(* Schneider Machine Expert - Basic project punya faris yang diomelin Ichsan Pan8, file version 1.7.0.0 *)
(* ProjectInformations: Name=New project *)

HARDWARE
  Cpu 0: TM221M16R/G
  EthernetConfiguration: NetworkName=M221, IpAllocationMode=FixedAddress, IpAddress=0.0.0.0, SubnetMask=0.0.0.0
  SerialLineConfiguration: Baud=Baud19200, Parity=ParityEven, DataBits=DataBits8, StopBits=StopBits1, PhysicalMedium=PhysicalMediumRs485, TransmissionMode=TransmissionModeModbusRtu, SlaveId=1, Addressing=SlaveAddressing
  MastTask: UsePeriodScanMode=false, PeriodScan=100
  FastTask: Period=255
  CpuBehavior: StartingMode=StartAsPreviousState, AutoSaveRamOnEeprom=true, WatchdogPeriod=250

SYMBOLS  (address, symbol, comment, settings)
  %M0         "manual"
  %M7         "auto"
  %I0.0       "Selektor"
  %I0.1       "SWITCH MANUAL"
  %I0.2       "Switch1"
  %I0.3       "Switch2"
  %I0.4       "Swutch3"
  %Q0.1       "Lampu1"
  %Q0.2       "Lampu2"

POU New POU
  (* SectionNumber=1 *)

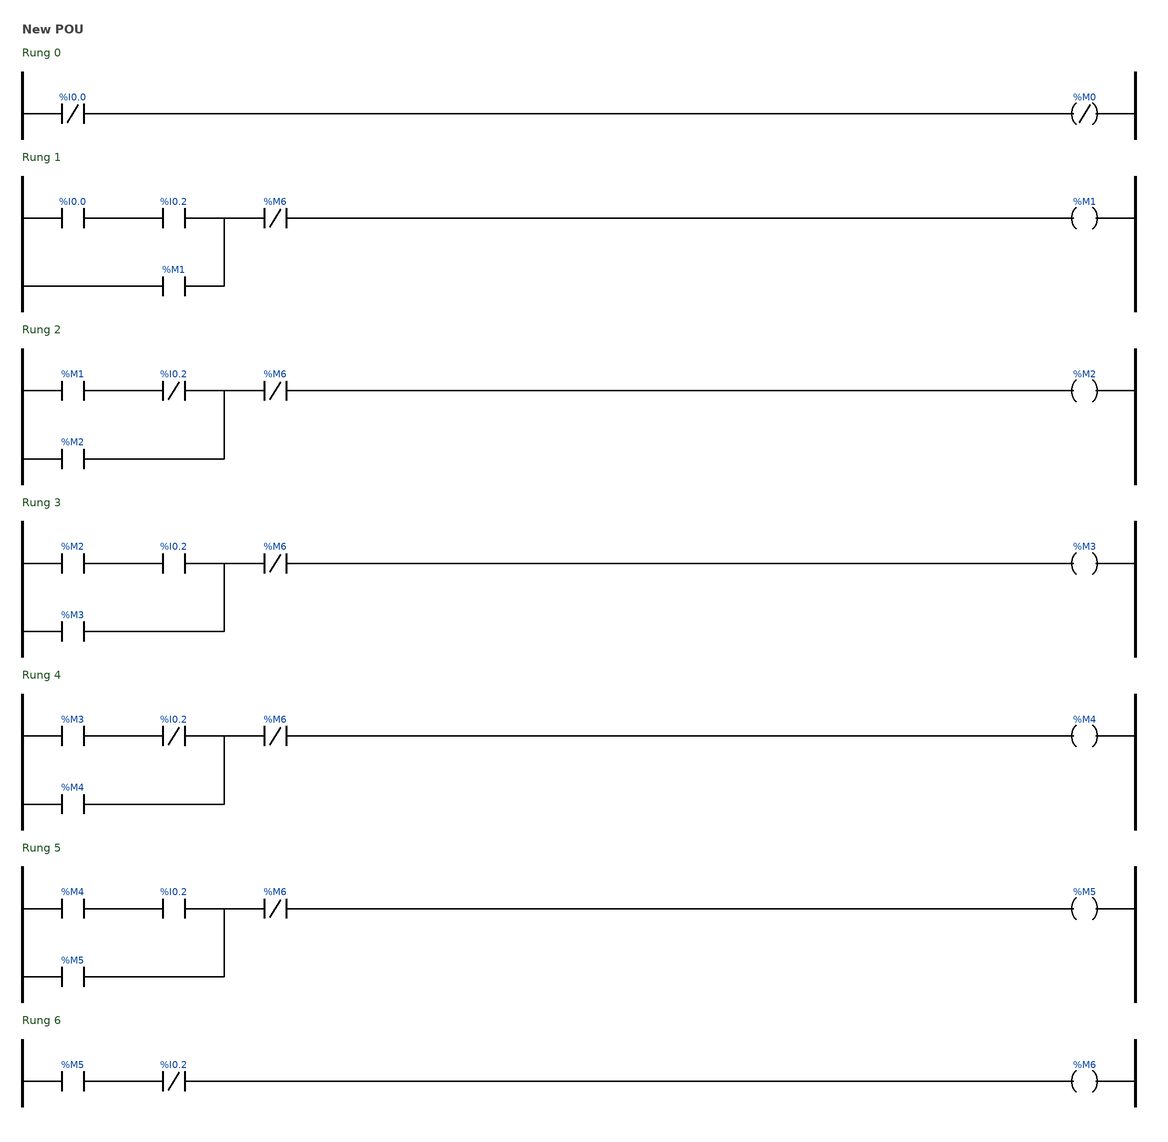

// Rung 0
  LDN %I0.0
  STN %M0
  // as ST:
  //   %M0 := NOT (NOT %I0.0);

// Rung 1
  LD %I0.0
  AND %I0.2
  OR %M1
  ANDN %M6
  ST %M1
  // as ST:
  //   %M1 := (%I0.0 AND %I0.2 OR %M1) AND NOT %M6;

// Rung 2
  LD %M1
  ANDN %I0.2
  OR %M2
  ANDN %M6
  ST %M2
  // as ST:
  //   %M2 := (%M1 AND NOT %I0.2 OR %M2) AND NOT %M6;

// Rung 3
  LD %M2
  AND %I0.2
  OR %M3
  ANDN %M6
  ST %M3
  // as ST:
  //   %M3 := (%M2 AND %I0.2 OR %M3) AND NOT %M6;

// Rung 4
  LD %M3
  ANDN %I0.2
  OR %M4
  ANDN %M6
  ST %M4
  // as ST:
  //   %M4 := (%M3 AND NOT %I0.2 OR %M4) AND NOT %M6;

// Rung 5
  LD %M4
  AND %I0.2
  OR %M5
  ANDN %M6
  ST %M5
  // as ST:
  //   %M5 := (%M4 AND %I0.2 OR %M5) AND NOT %M6;

// Rung 6
  LD %M5
  ANDN %I0.2
  ST %M6
  // as ST:
  //   %M6 := %M5 AND NOT %I0.2;

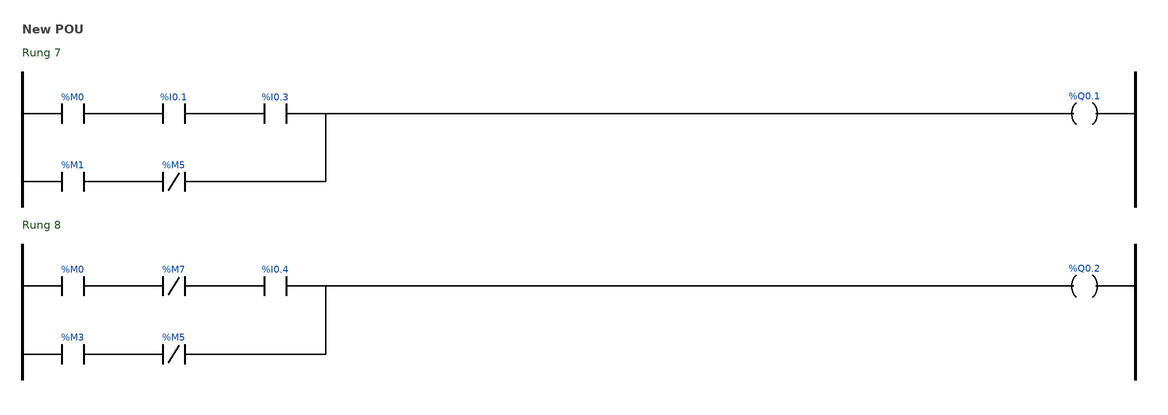

// Rung 7
  LD %M0
  AND %I0.1
  AND %I0.3
  OR( %M1
  ANDN %M5
  )
  ST %Q0.1
  // as ST:
  //   %Q0.1 := %M0 AND %I0.1 AND %I0.3 OR %M1 AND NOT %M5;

// Rung 8
  LD %M0
  ANDN %M7
  AND %I0.4
  OR( %M3
  ANDN %M5
  )
  ST %Q0.2
  // as ST:
  //   %Q0.2 := %M0 AND NOT %M7 AND %I0.4 OR %M3 AND NOT %M5;
